INTERFACE I_ForceableBOOL EXTENDS I_Bool

PROPERTY name : STRING
GET
END_GET
END_PROPERTY

PROPERTY path : STRING
GET
END_GET
END_PROPERTY

METHOD force
VAR_INPUT
    forcedValue : BOOL;
END_VAR
END_METHOD

METHOD release
END_METHOD

PROPERTY isForced : BOOL
GET
END_GET
END_PROPERTY

END_INTERFACE

(* stored: Version 1.1.0.1, ProductVersion 3.1.4026.18
   Itf I_ForceableBOOL: Id {e4d5f6a7-b8c9-0123-defa-234567890123}
   Property name: Id {11aa22bb-33cc-44dd-55ee-66ff77889900}
   Get Get: Id {22bb33cc-44dd-55ee-66ff-778899001122}
   Property path: Id {33cc44dd-55ee-66ff-7788-990011223344}
   Get Get: Id {44dd55ee-66ff-7788-9900-112233445566}
   Method force: Id {f5e6a7b8-c9d0-1234-efab-345678901234}
   Method release: Id {a6f7b8c9-d0e1-2345-fabc-456789012345}
   Property isForced: Id {b7a8c9d0-e1f2-3456-abcd-567890123456}
   Get Get: Id {c8b9d0e1-f2a3-4567-bcde-678901234567} *)
